FUNCTION_BLOCK FB_SoDuration_DB
VAR_INPUT
	udiDBID : UDINT := 1 ;
END_VAR

VAR_OUTPUT
	bBusy 		: BOOL;
	bDone		: BOOL;
	bError		: BOOL;
	udiErrId	: UDINT;
END_VAR

VAR
	// FBs
	FB_PLCDBCmdEvt_so_duration : FB_PLCDBCmdEvt(sNetID := '' , tTimeout := T#10S) ;
	
	// Vars
	stPara_so_duration 	: ARRAY[0..9] OF ST_ExpParameter ;
	iStep				: INT;
	iErrStep			: INT := 9000;
	
	// SQL Command
	
	(*
	sCmd_so_duration : STRING(1000) := '
		INSERT INTO [dbo].[so_duration] 
					([batch_start_time], [batch_end_time], [normal_complition], [batch_end_reason], [batch_end_reason_description], [employee_name_start_user], [employee_name_end_user], [so_number], [faam_id], [so_id]) 
		VALUES 		({dt_batch_start_time}, {dt_batch_end_time}, {b_normal_complition}, $'{wstr_batch_end_reason}$', $'{wstr_batch_end_reason_description}$', $'{wstr_employee_name_start_user}$', $'{wstr_employee_name_end_user}$', $'{str_so_number}$', $'{str_faam_id}$', {di_so_id}) ' ;
	*)
	
	
	sCmd_so_duration : STRING(1000) := '
		INSERT INTO [dbo].[so_duration] 
					([batch_start_time], [batch_end_time], [batch_end_reason], [batch_end_reason_description], [employee_name_start_user], [employee_name_end_user], [so_number], [faam_id], [so_id], [normal_complition]) 
		VALUES 		({dt_batch_start_time}, {dt_batch_end_time}, $'{wstr_batch_end_reason}$', $'{wstr_batch_end_reason_description}$', $'{wstr_employee_name_start_user}$', $'{wstr_employee_name_end_user}$', $'{str_so_number}$', $'{str_faam_id}$', {di_so_id}, {b_normal_complition}) ' ;
	
	
	
	// Time
	tStartTime	: TIME;
	tEndTime	: TIME;
	tDuration	: TIME;	
END_VAR

METHOD PRIVATE M_ClearStatus : BOOL
VAR_INPUT
END_VAR
bBusy := FALSE;
bDone := FALSE;
bError := FALSE;
udiErrId := 0;
END_METHOD

METHOD M_Reset : BOOL
VAR_INPUT
END_VAR
iStep := 0;
M_ClearStatus();
END_METHOD

METHOD PRIVATE M_SetBusy : BOOL
VAR_INPUT
END_VAR
bError := FALSE;
bBusy := TRUE;
bDone := FALSE;
END_METHOD

METHOD PRIVATE M_SetDone : BOOL
VAR_INPUT
END_VAR
bError := FALSE;
bBusy := FALSE;
bDone := TRUE;
END_METHOD

METHOD PRIVATE M_SetError : BOOL
VAR_INPUT
END_VAR
bError := TRUE;
bBusy := FALSE;
bDone := FALSE;
END_METHOD

METHOD Private M_SetSQLCmdPara : BOOL
VAR_INPUT
END_VAR
(*
stPara_so_duration[0].sParaName := 'dt_batch_start_time' ;
stPara_so_duration[0].eParaType := E_ExpParameterType.DateTime ;
stPara_so_duration[0].nParaSize := SIZEOF(ST_SoDuration.dtBatch_start_time) ;
stPara_so_duration[1].sParaName := 'dt_batch_end_time' ;
stPara_so_duration[1].eParaType := E_ExpParameterType.DateTime ;
stPara_so_duration[1].nParaSize := SIZEOF(ST_SoDuration.dtBatch_end_time) ;
stPara_so_duration[2].sParaName := 'b_normal_complition' ;
stPara_so_duration[2].eParaType := E_ExpParameterType.Boolean ;
stPara_so_duration[2].nParaSize := SIZEOF(ST_SoDuration.bNormal_complition) ;
stPara_so_duration[3].sParaName := 'wstr_batch_end_reason' ;
stPara_so_duration[3].eParaType := E_ExpParameterType.WSTRING_ ;
stPara_so_duration[3].nParaSize := SIZEOF(ST_SoDuration.wsBatch_end_reason) ;
stPara_so_duration[4].sParaName := 'wstr_batch_end_reason_description' ;
stPara_so_duration[4].eParaType := E_ExpParameterType.WSTRING_ ;
stPara_so_duration[4].nParaSize := SIZEOF(ST_SoDuration.wsBatch_end_reason_description) ;
stPara_so_duration[5].sParaName := 'wstr_employee_name_start_user' ;
stPara_so_duration[5].eParaType := E_ExpParameterType.WSTRING_ ;
stPara_so_duration[5].nParaSize := SIZEOF(ST_SoDuration.wsEmployee_name_start_user) ;
stPara_so_duration[6].sParaName := 'wstr_employee_name_end_user' ;
stPara_so_duration[6].eParaType := E_ExpParameterType.WSTRING_ ;
stPara_so_duration[6].nParaSize := SIZEOF(ST_SoDuration.wsEmployee_name_end_user) ;
stPara_so_duration[7].sParaName := 'str_so_number' ;
stPara_so_duration[7].eParaType := E_ExpParameterType.STRING_ ;
stPara_so_duration[7].nParaSize := SIZEOF(ST_SoDuration.sSo_number) ;
stPara_so_duration[8].sParaName := 'str_faam_id' ;
stPara_so_duration[8].eParaType := E_ExpParameterType.STRING_ ;
stPara_so_duration[8].nParaSize := SIZEOF(ST_SoDuration.sFaam_id) ;
stPara_so_duration[9].sParaName := 'di_so_id' ;
stPara_so_duration[9].eParaType := E_ExpParameterType.Int32 ;
stPara_so_duration[9].nParaSize := SIZEOF(ST_SoDuration.diSo_id) ;
*)


stPara_so_duration[0].sParaName := 'dt_batch_start_time' ;
stPara_so_duration[0].eParaType := E_ExpParameterType.DateTime ;
stPara_so_duration[0].nParaSize := SIZEOF(ST_SoDuration.dtBatch_start_time) ;
stPara_so_duration[1].sParaName := 'dt_batch_end_time' ;
stPara_so_duration[1].eParaType := E_ExpParameterType.DateTime ;
stPara_so_duration[1].nParaSize := SIZEOF(ST_SoDuration.dtBatch_end_time) ;
stPara_so_duration[2].sParaName := 'wstr_batch_end_reason' ;
stPara_so_duration[2].eParaType := E_ExpParameterType.WSTRING_ ;
stPara_so_duration[2].nParaSize := SIZEOF(ST_SoDuration.wsBatch_end_reason) ;
stPara_so_duration[3].sParaName := 'wstr_batch_end_reason_description' ;
stPara_so_duration[3].eParaType := E_ExpParameterType.WSTRING_ ;
stPara_so_duration[3].nParaSize := SIZEOF(ST_SoDuration.wsBatch_end_reason_description) ;
stPara_so_duration[4].sParaName := 'wstr_employee_name_start_user' ;
stPara_so_duration[4].eParaType := E_ExpParameterType.WSTRING_ ;
stPara_so_duration[4].nParaSize := SIZEOF(ST_SoDuration.wsEmployee_name_start_user) ;
stPara_so_duration[5].sParaName := 'wstr_employee_name_end_user' ;
stPara_so_duration[5].eParaType := E_ExpParameterType.WSTRING_ ;
stPara_so_duration[5].nParaSize := SIZEOF(ST_SoDuration.wsEmployee_name_end_user) ;
stPara_so_duration[6].sParaName := 'str_so_number' ;
stPara_so_duration[6].eParaType := E_ExpParameterType.STRING_ ;
stPara_so_duration[6].nParaSize := SIZEOF(ST_SoDuration.sSo_number) ;
stPara_so_duration[7].sParaName := 'str_faam_id' ;
stPara_so_duration[7].eParaType := E_ExpParameterType.STRING_ ;
stPara_so_duration[7].nParaSize := SIZEOF(ST_SoDuration.sFaam_id) ;
stPara_so_duration[8].sParaName := 'di_so_id' ;
stPara_so_duration[8].eParaType := E_ExpParameterType.Int32 ;
stPara_so_duration[8].nParaSize := SIZEOF(ST_SoDuration.diSo_id) ;
stPara_so_duration[9].sParaName := 'b_normal_complition' ;
stPara_so_duration[9].eParaType := E_ExpParameterType.Boolean ;
stPara_so_duration[9].nParaSize := SIZEOF(ST_SoDuration.bNormal_complition) ;


M_SetSQLCmdPara := TRUE;
END_METHOD

METHOD M_Upload : BOOL
VAR_INPUT
	stSoDuration : ST_SoDuration ;
END_VAR
VAR_INST
	ITF_TcMessage : Tc3_EventLogger.I_TcMessage;
END_VAR
CASE iStep OF
	0: 
		// SQLCmd的變數設定
		M_SetSQLCmdPara();
		
		tStartTime := TIME();
		M_SetBusy();
		iStep := iStep + 100;
		
	100:
		IF FB_PLCDBCmdEvt_so_duration.Execute
			(
				hDBID        := udiDBID ,
			 	pExpression  := ADR(sCmd_so_duration) , //SQL 指令的字串
			 	cbExpression := SIZEOF(sCmd_so_duration) ,
			 	pData        := ADR(stSoDuration) , //SQL 指令字串中的變數值，比如Keyword1數值是0，會帶入sCmd中的{Keyword}
			 	cbData       := SIZEOF(stSoDuration) ,
			 	pParameter   := ADR(stPara_so_duration) , //SQL 指令字串中的變數的類型，比如sParaName為'Keyword'
			 	cbParameter  := SIZEOF(stPara_so_duration) ,
			)
		THEN
			IF FB_PLCDBCmdEvt_so_duration.bError THEN // 異常
				ITF_TcMessage := FB_PLCDBCmdEvt_so_duration.ipTcResult;
				udiErrid := ITF_TcMessage.nEventId;	
				M_SetError();		
				iStep := iErrStep + 100;
			ELSE // 成功寫入
				M_Upload := TRUE;
				tEndTime := TIME();
				tDuration := tEndTime - tStartTime;
				M_SetDone();
				iStep := 0;
			END_IF
		END_IF

END_CASE
END_METHOD

END_FUNCTION_BLOCK

(* stored: Version 1.1.0.1, ProductVersion 3.1.4024.11
   POU FB_SoDuration_DB: Id {efa6f031-8e8e-42dc-8111-9c8ae84cc81a}, SpecialFunc None
   Method M_ClearStatus: Id {1d07091d-e126-4afd-9958-d1fd3fa02c83}
   Method M_Reset: Id {011604a9-1da2-4439-a5e4-f0066cbba774}
   Method M_SetBusy: Id {b9f85a6d-c8c3-4094-bbc5-d4015aad6fd6}
   Method M_SetDone: Id {b8d99cb6-b603-4a4b-96d2-b0fda4238352}
   Method M_SetError: Id {81997820-cee2-41ef-8510-54d265e92cb1}
   Method M_SetSQLCmdPara: Id {79546262-bc42-4529-aa7f-6b91ada57e13}
   Method M_Upload: Id {8b6a5a33-ceb5-4b05-9ca7-fa1c412aae8a} *)
